{region '#Template'}
	{attribute 'Category' := 'AC'}
	{attribute 'Version' := '0.0.1.0'}
	{attribute 'Tags' := 'AC, Aggregates, Cooler, Temperature'}
	{attribute 'Description' := 'Aggregat Kühler Temperatur mit Ventil	// Aggregate cooler temperature with valve'}
{endregion}
FUNCTION_BLOCK FB_BA_AC_ColT_02 EXTENDS FB_BA_AggregateB
VAR_INPUT
	fSpTSuA					: REAL;
	fTSuA					: REAL;
END_VAR
VAR_OUTPUT
	fPresentValue			: REAL;	
	bActiveSeqCtrl			: BOOL;
END_VAR
VAR_INPUT CONSTANT PERSISTENT
END_VAR
VAR_INPUT CONSTANT
	TFl						: FB_BA_SensorAnalog_IO;												
	TRt						: FB_BA_SensorAnalog_IO;			
	TSuACtrl				: FB_BA_AC_ColTSuACtrl;
	Vlv						: FB_BA_Vlv;
END_VAR
VAR		
END_VAR

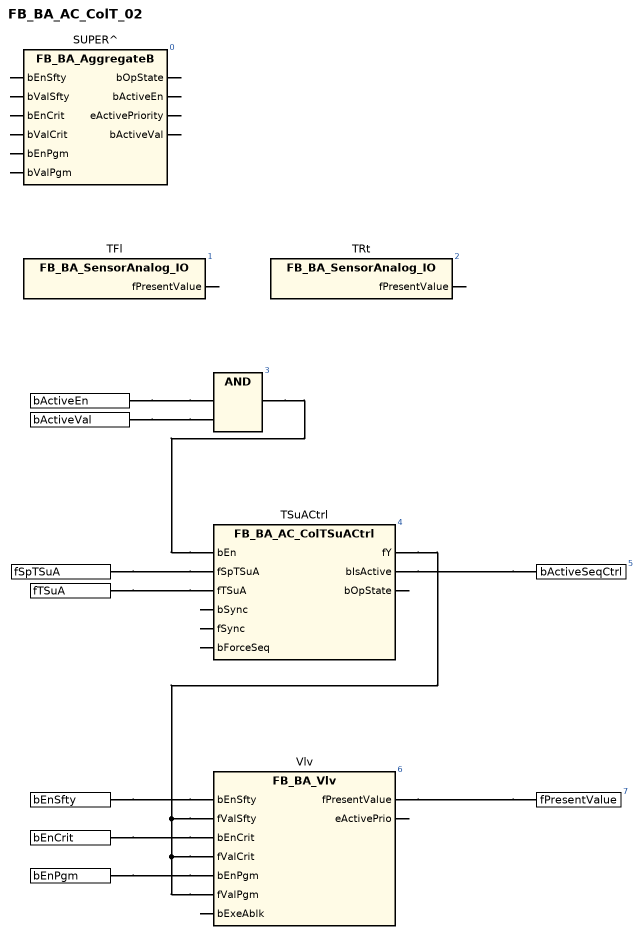
SUPER^(); // FB_BA_AggregateB
TFl(); // FB_BA_SensorAnalog_IO
TRt(); // FB_BA_SensorAnalog_IO
TSuACtrl(bEn := bActiveEn AND bActiveVal, fSpTSuA := fSpTSuA, fTSuA := fTSuA); // FB_BA_AC_ColTSuACtrl
bActiveSeqCtrl := TSuACtrl.bIsActive;
Vlv(
    bEnSfty := bEnSfty,
    fValSfty := TSuACtrl.fY,
    bEnCrit := bEnCrit,
    fValCrit := TSuACtrl.fY,
    bEnPgm := bEnPgm,
    fValPgm := TSuACtrl.fY); // FB_BA_Vlv
fPresentValue := Vlv.fPresentValue;

METHOD FB_init : BOOL
VAR_INPUT
	bInitRetains : BOOL; // if TRUE, the retain variables are initialized (warm start / cold start)
	bInCopyCode : BOOL;  // if TRUE, the instance afterwards gets moved into the copy code (online change)
END_VAR
TFl.iParent				:= THIS^;		
TFl.iLabel 				:= LblCmpAC.Cooler_TFl;	
TFl.sObjectName			:= '{Idx=41}';		
TFl.eDPADMode			:= E_BA_DPADMode.eInclude;															
TFl.MV.eUnit			:= E_BA_Unit.eTemperature_DegreesCelsius;
TFl.MV.eEnPlantLock		:= E_BA_LockPriority.eNoLock;
TFl.MV.fResolution 		:= 0.01;
TFl.MV.fScaleOffset 	:= 0; 

TRt.iParent				:= THIS^;		
TRt.iLabel 				:= LblCmpAC.Cooler_TRt;	
TRt.sObjectName			:= '{Idx=41}';		
TRt.eDPADMode			:= E_BA_DPADMode.eInclude;																											
TRt.MV.eUnit			:= E_BA_Unit.eTemperature_DegreesCelsius;
TRt.MV.eEnPlantLock		:= E_BA_LockPriority.eNoLock;
TRt.MV.fResolution 		:= 0.01;
TRt.MV.fScaleOffset 	:= 0;  

TSuACtrl.iParent		:= THIS^;	
TSuACtrl.iLabel			:= LblCmpAC.Cooler_TSuACtrl;
TSuACtrl.sObjectName	:= '{Idx=41}';										 
TSuACtrl.eDPADMode		:= E_BA_DPADMode.eInclude;								

Vlv.iParent				:= THIS^;
Vlv.iLabel				:= LblCmpAC.Cooler_Vlv;
Vlv.sObjectName			:= '{Idx=41}';										 
Vlv.eDPADMode			:= E_BA_DPADMode.eInclude;
END_METHOD

END_FUNCTION_BLOCK

(* stored: Version 1.1.0.1, ProductVersion 3.1.4024.6
   POU FB_BA_AC_ColT_02: Id {02596c09-d417-4f54-9e9e-8089c1b3e877}, SpecialFunc None
   Method FB_init: Id {b64f6103-0d34-457a-bb3c-2b6bc3ad8ec8} *)
